// TwinCAT 3 PLC project Untitled1
// ProgramVersion: 3.1.4022.2
// libraries:
//   Tc2_Standard, * (Beckhoff Automation GmbH)
//   Tc2_System, * (Beckhoff Automation GmbH)
//   Tc3_Module, * (Beckhoff Automation GmbH)
// project tree:
//   / PlcTask.TcTTO
//   POUs/ base.TcPOU, derived1.TcPOU, derived2.TcPOU, ITF.TcIO, MAIN.TcPOU

CONFIGURATION Untitled1
    RESOURCE PLC ON TwinCAT3
        TASK PlcTask(INTERVAL := T#10ms, PRIORITY := 20);
        PROGRAM MAIN WITH PlcTask : MAIN;
    END_RESOURCE
END_CONFIGURATION

// ---- POUs/ITF.TcIO
INTERFACE ITF

METHOD ITF_METH : STRING
VAR_INPUT
END_VAR
END_METHOD

END_INTERFACE

// ---- POUs/MAIN.TcPOU
PROGRAM MAIN
VAR
	anchor : POINTER TO base;
	itf_anchor : POINTER TO ITF;
	
	parent : base;
	child1 : derived1;
	child2 : derived2;

	output : string;
END_VAR


anchor := ADR(parent);
output := anchor^.METH();

anchor := ADR(child1);
output := anchor^.METH();

anchor := ADR(child2);
output := anchor^.METH();
//polymorphism is possible

//complition error
itf_anchor := ADR(child1);
output := itf_anchor^.ITF_METH();

itf_anchor := ADR(child2);
output := itf_anchor^.ITF_METH();

END_PROGRAM

// ---- POUs/base.TcPOU
FUNCTION_BLOCK base 
VAR_INPUT
END_VAR
VAR_OUTPUT
END_VAR
VAR
	field1 : INT := 555;
END_VAR

METHOD METH : STRING
VAR_INPUT
END_VAR
METH := 'base';
END_METHOD

END_FUNCTION_BLOCK

// ---- POUs/derived1.TcPOU
FUNCTION_BLOCK derived1 EXTENDS base implements itf
VAR_INPUT
END_VAR
VAR_OUTPUT
END_VAR
VAR
END_VAR

METHOD ITF_METH : STRING
VAR_INPUT
END_VAR
ITF_METH := 'derived1 itf method';
END_METHOD

METHOD METH : STRING
VAR_INPUT
END_VAR
METH := 'derived1';
END_METHOD

END_FUNCTION_BLOCK

// ---- POUs/derived2.TcPOU
FUNCTION_BLOCK derived2 EXTENDS base implements itf
VAR_INPUT
END_VAR
VAR_OUTPUT
END_VAR
VAR
END_VAR

METHOD ITF_METH : STRING
VAR_INPUT
END_VAR
ITF_METH := 'derived2 itf method';
END_METHOD

METHOD METH : string
VAR_INPUT
END_VAR
METH := 'derived2';
END_METHOD

END_FUNCTION_BLOCK
